// TIA Portal V20 export
TYPE "HMI_CntOhSc"
   STRUCT
      OnOp : Bool := FALSE;   // 1=On Mode: On Mode by Operator
      OosOp : Bool := FALSE;   // 1=Oos Mode: Oos Mode by Operator
      OffOp : Bool := TRUE;   // 1= Counter Off by Operator
      UpOp : Bool := FALSE;   // 1= Counter Up by Operator
      ResetOp : Bool := FALSE;   // 1= Counter Reset by Operator
      HrsHi1Lim : DInt := 2280;   // Hours, High Limit 195 days
      HrsHi2Lim : DInt := 2160;   // Hours, High Limit 290 days
      CntHi1Lim : DInt := 95;   // Counter, High Limit 1
      CntHi2Lim : DInt := 90;   // Counter, High Limit 2
      HrsOpHiScale : DInt := 2400;   // Operation Hours Bar Display High Value100 Days
      HrsOpLoScale : DInt := 0;   // Operation Hours Bar Display Low Value
      CntOpHiScale : DInt := 100;   // Cnt - Bar Display Limits for OS High Value
      CntOpLoScale : DInt := 0;   // Cnt - Bar Display Limits for OS Low Value
      CntUnit : Int := 0;   // Unit of Cnt
      DeviceOn { ExternalWritable := 'False'} : Bool;   // 1= Device On
      CountMode { ExternalWritable := 'False'} : Int := 0;   // Counting Mode; 0=Off,1=Up
      Days { ExternalWritable := 'False'} : Int := 0;   // Operating Days
      Hours { ExternalWritable := 'False'} : Int := 0;   // Operating Hours
      TimeHours { ExternalWritable := 'False'} : DInt := 0;   // Operating Time [In Hours]
      Cnt { ExternalWritable := 'False'} : DInt := 0;   // Counter Value
      OS_PermOut { ExternalWritable := 'False'} : DWord := 16#FFFF_FFFF;   // Operator Permission: Output for OS
      OS_PermLog { ExternalWritable := 'False'} : DWord := 16#FFFF_FFFF;   // Operator Permission: Output for OS
      OpSt_Out { ExternalWritable := 'False'} : DWord := 16#0000_0000;   // Enabled operator stations
      ST_Worst { ExternalWritable := 'False'} : Byte := 16#80;   // Worst Signal Status
      Status1 { ExternalWritable := 'False'} : DWord := 16#0000_0000;   // Status1 Word
      Status2 { ExternalWritable := 'False'} : DWord := 16#0000_0000;   // Status2 Word
   END_STRUCT;
END_TYPE
